// TIA Portal V20 export
// export: Created 2025-12-01T14:57:12.6203734Z, ExportSetting None, DisplayName Totally Integrated Automation Portal, DisplayVersion V20 Update 3, DisplayName TIA Portal Openness, DisplayVersion V20 Update 3, DisplayName TIA Portal Version Control Interface, DisplayVersion V20 Update 3, DisplayName STEP 7 Professional, DisplayVersion V20 Update 3, DisplayName STEP 7 Safety, DisplayVersion V20 Update 2, DisplayName WinCC Basic/Comfort/Advanced, DisplayVersion V20 Update 3, DisplayName WinCC Professional, DisplayVersion V20 Update 3, DisplayName WinCC Unified, DisplayVersion V20 Update 3
FUNCTION "FC994_CTRL_VAR_Lenze_i550_ES" : Void   // FC994, LAD
{ S7_Optimized_Access := 'TRUE' }
NAME : 20181121
VERSION : 1.0
// stored: AutoNumber false, SetENOAutomatically false
   VAR_INPUT
      Avance : Bool;
      Retroceso : Bool;
      Rearme : Bool;
      Velocidad : Int;   // La velocidad es un entero que tiene que se 1, 2 o 3
      Sentido_Giro : Bool;
   END_VAR
   VAR_OUTPUT
      Av_Ret_Tx : Bool;   // Marca para informar de que se esta moviendo el variador
      Run : Bool;   // Señal de avance
      Reverse : Bool;   // Señal de Retroceso
      Vel_1 : Bool;
      Vel_2 : Bool;
   END_VAR
   VAR_TEMP   // added for the SCL form of the ladder/FBD networks
      _w1 : Bool;
   END_VAR
BEGIN

REGION Network 1: Activación del RUN del i550 a E/S - DI01
   // Siempre hay que activar el RUN del variador. Hagamos AVANCE o RETROCESO el RUN siempre activo
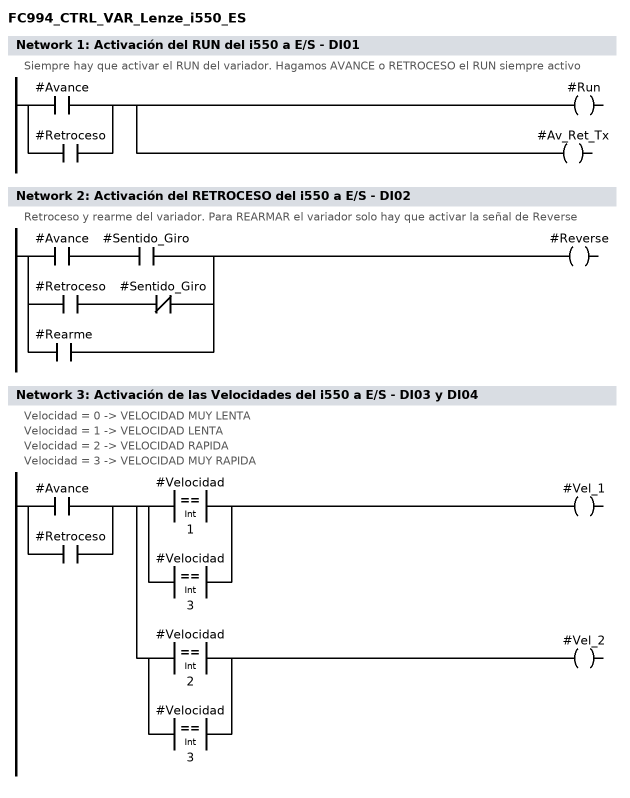
   RUNG wire#powerrail
      Contact( #Avance )
      wire#w1
      Coil( #Run )
   END_RUNG
   RUNG wire#powerrail
      Contact( #Retroceso )
   END_RUNG wire#w1
   RUNG wire#w1
      Coil( #Av_Ret_Tx )
   END_RUNG
   // the same network as SCL:
   #Run := #Avance OR #Retroceso;
   #Av_Ret_Tx := #Run;
END_REGION

REGION Network 2: Activación del RETROCESO del i550 a E/S - DI02
   // Retroceso y rearme del variador. Para REARMAR el variador solo hay que activar la señal de Reverse
   RUNG wire#powerrail
      Contact( #Avance )
      Contact( #Sentido_Giro )
      wire#w1
      Coil( #Reverse )
   END_RUNG
   RUNG wire#powerrail
      Contact( #Retroceso )
      I_Contact( #Sentido_Giro )
   END_RUNG wire#w1
   RUNG wire#powerrail
      Contact( #Rearme )
   END_RUNG wire#w1
   // the same network as SCL:
   #Reverse := (#Avance AND #Sentido_Giro) OR (#Retroceso AND NOT #Sentido_Giro) OR #Rearme;
END_REGION

REGION Network 3: Activación de las Velocidades del i550 a E/S - DI03 y DI04
   // Velocidad = 0 -> VELOCIDAD MUY LENTA
   // Velocidad = 1 -> VELOCIDAD LENTA
   // Velocidad = 2 -> VELOCIDAD RAPIDA
   // Velocidad = 3 -> VELOCIDAD MUY RAPIDA
   RUNG wire#powerrail
      Contact( #Avance )
      wire#w1
      { S7_Templates := "SrcType := Int" } EQ_Contact(in1 := #Velocidad, in2 := 1)
      wire#w2
      Coil( #Vel_1 )
   END_RUNG
   RUNG wire#powerrail
      Contact( #Retroceso )
   END_RUNG wire#w1
   RUNG wire#w1
      { S7_Templates := "SrcType := Int" } EQ_Contact(in1 := #Velocidad, in2 := 3)
   END_RUNG wire#w2
   RUNG wire#w1
      { S7_Templates := "SrcType := Int" } EQ_Contact(in1 := #Velocidad, in2 := 2)
      wire#w3
      Coil( #Vel_2 )
   END_RUNG
   RUNG wire#w1
      { S7_Templates := "SrcType := Int" } EQ_Contact(in1 := #Velocidad, in2 := 3)
   END_RUNG wire#w3
   // the same network as SCL:
   #_w1 := #Avance OR #Retroceso;
   #Vel_1 := #_w1 AND ((#Velocidad = 1) OR (#Velocidad = 3));
   #Vel_2 := #_w1 AND ((#Velocidad = 2) OR (#Velocidad = 3));
END_REGION
END_FUNCTION
